TYPE ST_ReportInfo_CUL :
STRUCT
	reportName        : STRING;
    reoportSubName    : STRING;
    reportDate        : STRING;
    systemID          : STRING;
    databaseName      : STRING;
    page              : STRING;
    printedBy         : STRING;
	fileName		  : STRING;
END_STRUCT
END_TYPE

(* stored: Version 1.1.0.1, ProductVersion 3.1.4024.12
   DUT ST_ReportInfo_CUL: Id {492807dc-ab2e-4d1a-b732-7e3d7c278165} *)
